FUNCTION_BLOCK FILE_WRITER_1 (* Writes equation coeficients to a file (1 coef) *)
  (* Standard: 61499-2 *)
  (* Version 1.0, 21-03-12, GASR, Universidade do Estado de Santa Catarina *)
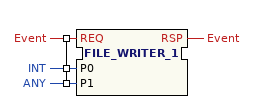
  EVENT_INPUT
    REQ WITH P0, P1; (* Request file storage *)
  END_EVENT
  EVENT_OUTPUT
    RSP; (* Finished operation *)
  END_EVENT
  VAR_INPUT
    P0 : INT; (* Process/equation id *)
    P1 : ANY; (* Coeficient 1 *)
  END_VAR
  SERVICE FILE_WRITER_1/MACHINE (* Coeficient file storage service *)
    SEQUENCE normal_establishment
      FILE_WRITER_1.REQ(P0,P1) -> MACHINE.write-file();
      MACHINE.response() -> FILE_WRITER_1.RSP();
    END_SEQUENCE
  END_SERVICE
END_FUNCTION_BLOCK
